// TIA Portal V15.1 export
// export: Created 2026-01-15T16:29:48.1018365Z, ExportSetting WithDefaults, WithReadOnly, DisplayName Totally Integrated Automation Portal, DisplayVersion V15.1 Update 8, DisplayName TIA Portal Openness, DisplayVersion V15.1 Update 8, DisplayName STEP 7 Professional, DisplayVersion V15.1 Update 8, DisplayName WinCC Advanced, DisplayVersion V15.1 Update 8
FUNCTION "FCXL_IND_AGG4" : Void   // FC23, LAD
{ S7_Optimized_Access := 'TRUE' }
VERSION : 0.1
// stored: AutoNumber true, CodeModifiedDate 2026-01-15T16:25:53.5191681Z, CompileDate 2026-01-15T16:25:53.5611578Z, CreationDate 2026-01-15T16:24:02.4619467Z, HandleErrorsWithinBlock false, InterfaceModifiedDate 2026-01-11T04:48:18.8495033Z, IsConsistent true, IsIECCheckEnabled false, IsKnowHowProtected false, IsWriteProtected false, LibraryConformanceStatus Error: The block contains calls of single instances. Warning: The object contains access to global data blocks. Warning: The block contains direct access to inputs, outputs, bit memories, indirect access to the registry or indirect access to external memory areas that are unknown at the time of compilation., ModifiedDate 2026-01-15T16:25:53.5191681Z, ParameterModified 2026-01-11T04:48:18.8495033Z, PLCSimAdvancedSupport false, SetENOAutomatically False, StructureModified 2026-01-11T04:48:18.8495033Z, UDAEnableTagReadback false
   VAR_TEMP   // added for the SCL form of the ladder/FBD networks
      _w1 : Bool;
      _w2 : Bool;
      _w3 : Bool;
   END_VAR
BEGIN

REGION Network 1: Cân độc lập AGG4 Full
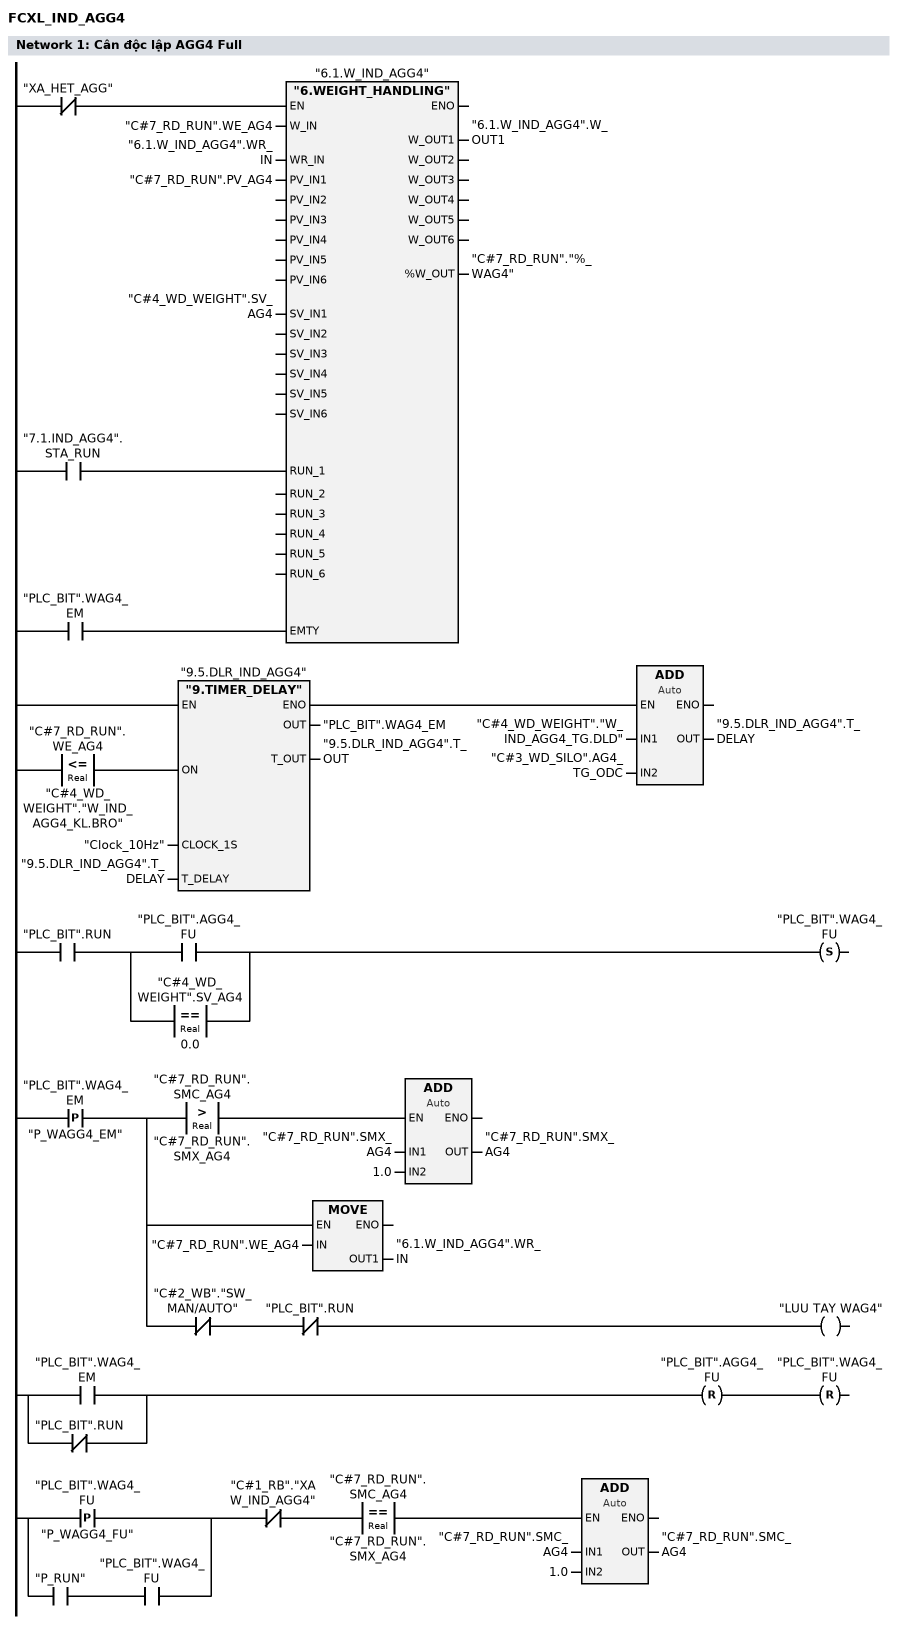
   RUNG wire#powerrail
      I_Contact( "XA_HET_AGG" )
      "6.1.W_IND_AGG4"(RUN_1 := wire#w1, EMTY := wire#w2, W_IN := "C#7_RD_RUN".WE_AG4, WR_IN := "6.1.W_IND_AGG4".WR_IN, PV_IN1 := "C#7_RD_RUN".PV_AG4, PV_IN2 :=, PV_IN3 :=, PV_IN4 :=, PV_IN5 :=, PV_IN6 :=, SV_IN1 := "C#4_WD_WEIGHT".SV_AG4, SV_IN2 :=, SV_IN3 :=, SV_IN4 :=, SV_IN5 :=, SV_IN6 :=, RUN_2 :=, RUN_3 :=, RUN_4 :=, RUN_5 :=, RUN_6 :=, W_OUT1 => "6.1.W_IND_AGG4".W_OUT1, W_OUT2 =>, W_OUT3 =>, W_OUT4 =>, W_OUT5 =>, W_OUT6 =>, "%W_OUT" => "C#7_RD_RUN"."%_WAG4")
   END_RUNG
   RUNG wire#powerrail
      Contact( "7.1.IND_AGG4".STA_RUN )
   END_RUNG wire#w1
   RUNG wire#powerrail
      Contact( "PLC_BIT".WAG4_EM )
   END_RUNG wire#w2
   RUNG wire#powerrail
      "9.5.DLR_IND_AGG4"(ON := wire#w3, CLOCK_1S := "Clock_10Hz", T_DELAY := "9.5.DLR_IND_AGG4".T_DELAY, OUT => "PLC_BIT".WAG4_EM, T_OUT => "9.5.DLR_IND_AGG4".T_OUT)
      Add(in1 := "C#4_WD_WEIGHT"."W_IND_AGG4_TG.DLD", in2 := "C#3_WD_SILO".AG4_TG_ODC, out => "9.5.DLR_IND_AGG4".T_DELAY)
   END_RUNG
   RUNG wire#powerrail
      { S7_Templates := "SrcType := Real" } LE_Contact(in1 := "C#7_RD_RUN".WE_AG4, in2 := "C#4_WD_WEIGHT"."W_IND_AGG4_KL.BRO")
   END_RUNG wire#w3
   RUNG wire#powerrail
      Contact( "PLC_BIT".RUN )
      wire#w4
      Contact( "PLC_BIT".AGG4_FU )
      wire#w5
      S_Coil( "PLC_BIT".WAG4_FU )
   END_RUNG
   RUNG wire#w4
      { S7_Templates := "SrcType := Real" } EQ_Contact(in1 := "C#4_WD_WEIGHT".SV_AG4, in2 := 0.0)
   END_RUNG wire#w5
   RUNG wire#powerrail
      P_Contact(operand := "PLC_BIT".WAG4_EM, bit := "P_WAGG4_EM")
      wire#w6
      { S7_Templates := "SrcType := Real" } GT_Contact(in1 := "C#7_RD_RUN".SMC_AG4, in2 := "C#7_RD_RUN".SMX_AG4)
      Add(in1 := "C#7_RD_RUN".SMX_AG4, in2 := 1.0, out => "C#7_RD_RUN".SMX_AG4)
   END_RUNG
   RUNG wire#w6
      Move(in := "C#7_RD_RUN".WE_AG4, out1 => "6.1.W_IND_AGG4".WR_IN)
   END_RUNG
   RUNG wire#w6
      I_Contact( "C#2_WB"."SW_MAN/AUTO" )
      I_Contact( "PLC_BIT".RUN )
      Coil( "LUU TAY WAG4" )
   END_RUNG
   RUNG wire#powerrail
      Contact( "PLC_BIT".WAG4_EM )
      wire#w7
      R_Coil( "PLC_BIT".AGG4_FU )
      R_Coil( "PLC_BIT".WAG4_FU )
   END_RUNG
   RUNG wire#powerrail
      I_Contact( "PLC_BIT".RUN )
   END_RUNG wire#w7
   RUNG wire#powerrail
      P_Contact(operand := "PLC_BIT".WAG4_FU, bit := "P_WAGG4_FU")
      wire#w8
      I_Contact( "C#1_RB"."XA W_IND_AGG4" )
      { S7_Templates := "SrcType := Real" } EQ_Contact(in1 := "C#7_RD_RUN".SMC_AG4, in2 := "C#7_RD_RUN".SMX_AG4)
      Add(in1 := "C#7_RD_RUN".SMC_AG4, in2 := 1.0, out => "C#7_RD_RUN".SMC_AG4)
   END_RUNG
   RUNG wire#powerrail
      Contact( "P_RUN" )
      Contact( "PLC_BIT".WAG4_FU )
   END_RUNG wire#w8
   // the same network as SCL:
   IF NOT "XA_HET_AGG" THEN
       "6.1.W_IND_AGG4"(W_IN := "C#7_RD_RUN".WE_AG4,   // "6.WEIGHT_HANDLING"
                        WR_IN := "6.1.W_IND_AGG4".WR_IN,
                        PV_IN1 := "C#7_RD_RUN".PV_AG4,
                        SV_IN1 := "C#4_WD_WEIGHT".SV_AG4,
                        RUN_1 := "7.1.IND_AGG4".STA_RUN,
                        EMTY := "PLC_BIT".WAG4_EM,
                        W_OUT1 => "6.1.W_IND_AGG4".W_OUT1,
                        "%W_OUT" => "C#7_RD_RUN"."%_WAG4");
   END_IF;
   "9.5.DLR_IND_AGG4"(ON := "C#7_RD_RUN".WE_AG4 <= "C#4_WD_WEIGHT"."W_IND_AGG4_KL.BRO",   // "9.TIMER_DELAY"
                      CLOCK_1S := "Clock_10Hz",
                      T_DELAY := "9.5.DLR_IND_AGG4".T_DELAY,
                      OUT => "PLC_BIT".WAG4_EM,
                      T_OUT => "9.5.DLR_IND_AGG4".T_OUT,
                      ENO => #_w1);
   IF #_w1 THEN
       "9.5.DLR_IND_AGG4".T_DELAY := "C#4_WD_WEIGHT"."W_IND_AGG4_TG.DLD" + "C#3_WD_SILO".AG4_TG_ODC;
   END_IF;
   IF "PLC_BIT".RUN AND ("PLC_BIT".AGG4_FU OR ("C#4_WD_WEIGHT".SV_AG4 = 0.0)) THEN
       "PLC_BIT".WAG4_FU := TRUE;
   END_IF;
   #_w2 := "PLC_BIT".WAG4_EM AND NOT "P_WAGG4_EM";   // rising edge of "PLC_BIT".WAG4_EM
   "P_WAGG4_EM" := "PLC_BIT".WAG4_EM;
   IF #_w2 AND ("C#7_RD_RUN".SMC_AG4 > "C#7_RD_RUN".SMX_AG4) THEN
       "C#7_RD_RUN".SMX_AG4 := "C#7_RD_RUN".SMX_AG4 + 1.0;
   END_IF;
   IF #_w2 THEN "6.1.W_IND_AGG4".WR_IN := "C#7_RD_RUN".WE_AG4; END_IF;
   "LUU TAY WAG4" := #_w2 AND NOT "C#2_WB"."SW_MAN/AUTO" AND NOT "PLC_BIT".RUN;
   IF "PLC_BIT".WAG4_EM OR NOT "PLC_BIT".RUN THEN
       "PLC_BIT".AGG4_FU := FALSE;
       "PLC_BIT".WAG4_FU := FALSE;
   END_IF;
   #_w3 := "PLC_BIT".WAG4_FU AND NOT "P_WAGG4_FU";   // rising edge of "PLC_BIT".WAG4_FU
   "P_WAGG4_FU" := "PLC_BIT".WAG4_FU;
   IF (#_w3 OR ("P_RUN" AND "PLC_BIT".WAG4_FU)) AND NOT "C#1_RB"."XA W_IND_AGG4" AND ("C#7_RD_RUN".SMC_AG4 = "C#7_RD_RUN".SMX_AG4) THEN
       "C#7_RD_RUN".SMC_AG4 := "C#7_RD_RUN".SMC_AG4 + 1.0;
   END_IF;
END_REGION
END_FUNCTION
